// TIA Portal V17 export
// export: Created 2023-12-22T15:02:58.5343493Z, ExportSetting WithDefaults, DisplayName Totally Integrated Automation Portal, DisplayVersion V17, DisplayName TIA Portal Openness, DisplayVersion V17, DisplayName TIA Portal Version Control Interface, DisplayVersion V17, DisplayName STEP 7 Professional, DisplayVersion V17, DisplayName STEP 7 Safety, DisplayVersion V17, DisplayName WinCC Advanced, DisplayVersion V17
ORGANIZATION_BLOCK "Main"   // OB1, LAD, ProgramCycle
TITLE = "Main Program Sweep (Cycle)"
{ S7_Optimized_Access := 'TRUE' }
VERSION : 0.1
// stored: AutoNumber true, IsIECCheckEnabled false, SetENOAutomatically false
   VAR_INPUT
      Initial_Call : Bool;   // Initial call of this OB
      Remanence : Bool;   // =True, if remanent data are available
   END_VAR
   VAR_TEMP   // added for the SCL form of the ladder/FBD networks
      _w1 : Bool;
      _w2 : Bool;
      _w3 : Bool;
      _w4 : Bool;
   END_VAR
BEGIN

REGION Network 1
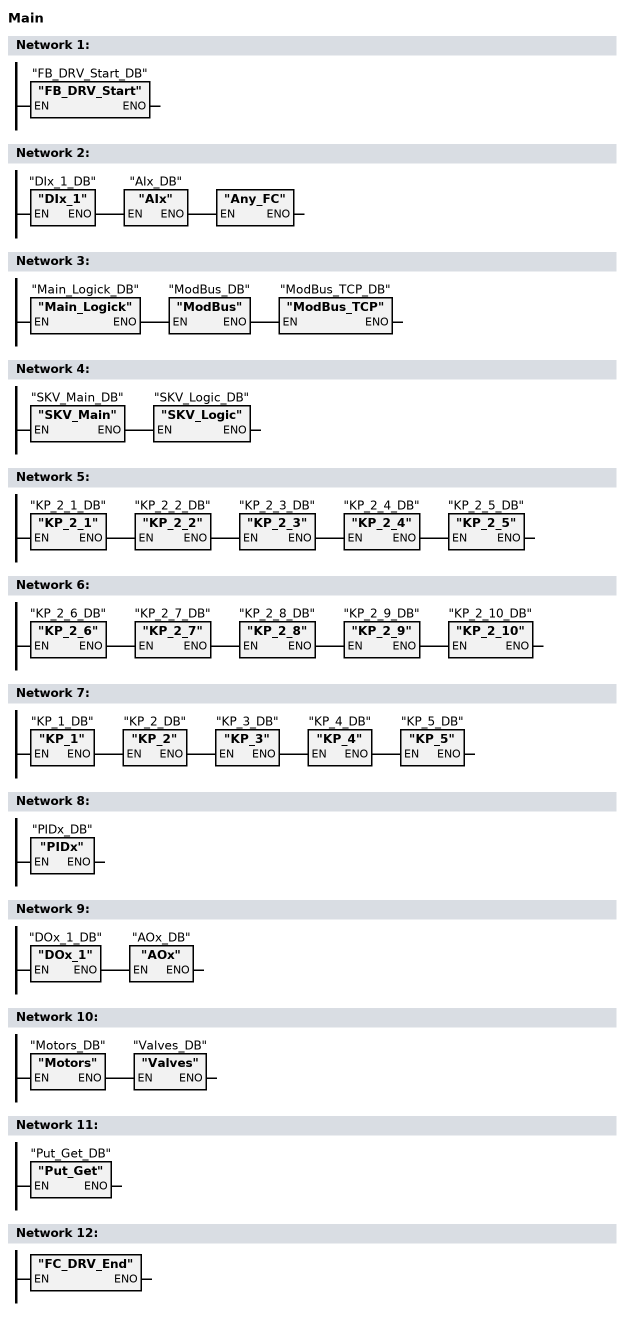
   RUNG wire#powerrail
      "FB_DRV_Start_DB"()
   END_RUNG
   // the same network as SCL:
   "FB_DRV_Start_DB"();   // "FB_DRV_Start"
END_REGION

REGION Network 2
   RUNG wire#powerrail
      "DIx_1_DB"()
      "AIx_DB"()
      "Any_FC"()
   END_RUNG
   // the same network as SCL:
   "DIx_1_DB"(ENO => #_w1);   // "DIx_1"
   "AIx_DB"(EN := #_w1, ENO => #_w2);   // "AIx"
   IF #_w2 THEN "Any_FC"(); END_IF;
END_REGION

REGION Network 3
   RUNG wire#powerrail
      "Main_Logick_DB"()
      "ModBus_DB"()
      "ModBus_TCP_DB"()
   END_RUNG
   // the same network as SCL:
   "Main_Logick_DB"(ENO => #_w1);   // "Main_Logick"
   "ModBus_DB"(EN := #_w1, ENO => #_w2);   // "ModBus"
   IF #_w2 THEN
       "ModBus_TCP_DB"();   // "ModBus_TCP"
   END_IF;
END_REGION

REGION Network 4
   RUNG wire#powerrail
      "SKV_Main_DB"()
      "SKV_Logic_DB"()
   END_RUNG
   // the same network as SCL:
   "SKV_Main_DB"(ENO => #_w1);   // "SKV_Main"
   IF #_w1 THEN
       "SKV_Logic_DB"();   // "SKV_Logic"
   END_IF;
END_REGION

REGION Network 5
   RUNG wire#powerrail
      "KP_2_1_DB"()
      "KP_2_2_DB"()
      "KP_2_3_DB"()
      "KP_2_4_DB"()
      "KP_2_5_DB"()
   END_RUNG
   // the same network as SCL:
   "KP_2_1_DB"(ENO => #_w1);   // "KP_2_1"
   "KP_2_2_DB"(EN := #_w1, ENO => #_w2);   // "KP_2_2"
   "KP_2_3_DB"(EN := #_w2, ENO => #_w3);   // "KP_2_3"
   "KP_2_4_DB"(EN := #_w3, ENO => #_w4);   // "KP_2_4"
   IF #_w4 THEN
       "KP_2_5_DB"();   // "KP_2_5"
   END_IF;
END_REGION

REGION Network 6
   RUNG wire#powerrail
      "KP_2_6_DB"()
      "KP_2_7_DB"()
      "KP_2_8_DB"()
      "KP_2_9_DB"()
      "KP_2_10_DB"()
   END_RUNG
   // the same network as SCL:
   "KP_2_6_DB"(ENO => #_w1);   // "KP_2_6"
   "KP_2_7_DB"(EN := #_w1, ENO => #_w2);   // "KP_2_7"
   "KP_2_8_DB"(EN := #_w2, ENO => #_w3);   // "KP_2_8"
   "KP_2_9_DB"(EN := #_w3, ENO => #_w4);   // "KP_2_9"
   IF #_w4 THEN
       "KP_2_10_DB"();   // "KP_2_10"
   END_IF;
END_REGION

REGION Network 7
   RUNG wire#powerrail
      "KP_1_DB"()
      "KP_2_DB"()
      "KP_3_DB"()
      "KP_4_DB"()
      "KP_5_DB"()
   END_RUNG
   // the same network as SCL:
   "KP_1_DB"(ENO => #_w1);   // "KP_1"
   "KP_2_DB"(EN := #_w1, ENO => #_w2);   // "KP_2"
   "KP_3_DB"(EN := #_w2, ENO => #_w3);   // "KP_3"
   "KP_4_DB"(EN := #_w3, ENO => #_w4);   // "KP_4"
   IF #_w4 THEN
       "KP_5_DB"();   // "KP_5"
   END_IF;
END_REGION

REGION Network 8
   RUNG wire#powerrail
      "PIDx_DB"()
   END_RUNG
   // the same network as SCL:
   "PIDx_DB"();   // "PIDx"
END_REGION

REGION Network 9
   RUNG wire#powerrail
      "DOx_1_DB"()
      "AOx_DB"()
   END_RUNG
   // the same network as SCL:
   "DOx_1_DB"(ENO => #_w1);   // "DOx_1"
   IF #_w1 THEN
       "AOx_DB"();   // "AOx"
   END_IF;
END_REGION

REGION Network 10
   RUNG wire#powerrail
      "Motors_DB"()
      "Valves_DB"()
   END_RUNG
   // the same network as SCL:
   "Motors_DB"(ENO => #_w1);   // "Motors"
   IF #_w1 THEN
       "Valves_DB"();   // "Valves"
   END_IF;
END_REGION

REGION Network 11
   RUNG wire#powerrail
      "Put_Get_DB"()
   END_RUNG
   // the same network as SCL:
   "Put_Get_DB"();   // "Put_Get"
END_REGION

REGION Network 12
   RUNG wire#powerrail
      "FC_DRV_End"()
   END_RUNG
   // the same network as SCL:
   "FC_DRV_End"();
END_REGION
END_ORGANIZATION_BLOCK
